FUNCTION_BLOCK FB_B IMPLEMENTS I_Name

VAR
    sVar2 : STRING := 'My name is B.'; 
END_VAR

{warning 'add property implementation'}
PROPERTY Name : STRING
GET
Name := sVar2;
END_GET
SET
sVar2 := Name;
END_SET
END_PROPERTY

END_FUNCTION_BLOCK

(* stored: Version 1.1.0.1, ProductVersion 3.1.4024.12
   POU FB_B: Id {1bd7c13a-1fb6-4420-b879-ff19c699f04a}, SpecialFunc None
   Property Name: Id {c99d6969-be3c-49de-bbda-2cd6a9cfa8fe}
   Get Get: Id {e93c5f2c-d5ac-4759-9b0d-09ce616a7887}
   Set Set: Id {6dbbd0c9-a124-4ac6-8301-b5dbedc9f0a3} *)
